(* Logix 5000 project; controller MetsoFilter vendor 1 type 14 code 106 rev 32.11; software revision 32.00; part 4 of 4 *)
(* tags used below, declared in another part *)
   AlwaysOff : BOOL;   // Always Off Bit
(* MainProgram, continued *)

ROUTINE MainRoutine   (* ladder *)
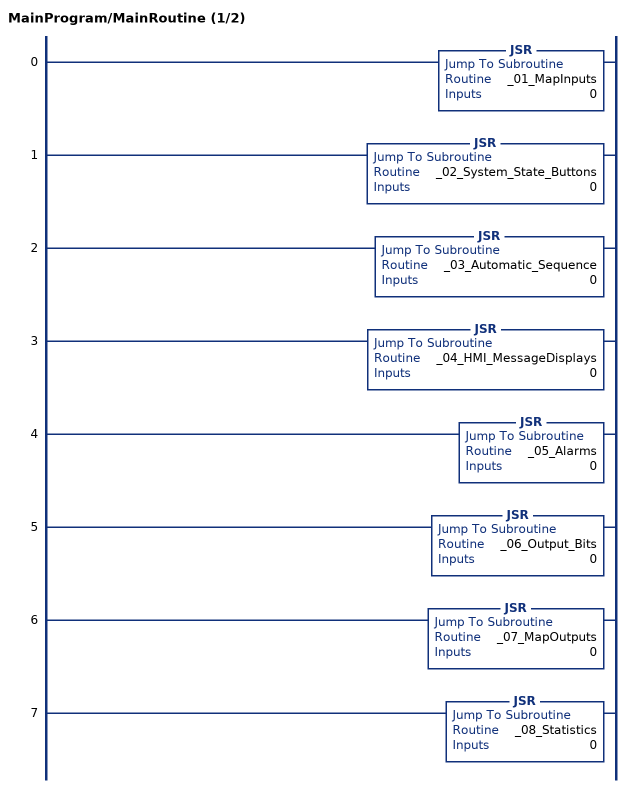
   0: JSR(_01_MapInputs,0);
   1: JSR(_02_System_State_Buttons,0);
   2: JSR(_03_Automatic_Sequence,0);
   3: JSR(_04_HMI_MessageDisplays,0);
   4: JSR(_05_Alarms,0);
   5: JSR(_06_Output_Bits,0);
   6: JSR(_07_MapOutputs,0);
   7: JSR(_08_Statistics,0);
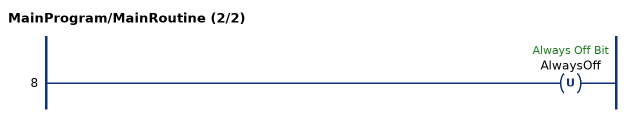
   8: OTU(AlwaysOff);
END_ROUTINE
END_PROGRAM
